{attribute addProperty BoxType "EL9222-4433-0018"}
{attribute addProperty Id "OCP_Inputs_ChannelAT %I*ARRAY[0..1] OF OCP_Inputs_Channel_FE08AF3C6480OCP_Outputs_ChannelAT %Q*ARRAY[0..1] OF OCP_Outputs_Channel_F330A9163240WcStateAT %I*WcState_98A4DF7520.250InfoDataAT %I*InfoData_BC63D37F80100"}
{attribute addProperty CRC "2874621807"}
{attribute addProperty SizeInBites "178"}
{attribute addProperty SizeInBytes "22.25"}
TYPE EL9222_58483589 :
STRUCT
	{attribute addProperty Name "OCP_Inputs_Channel"}
	OCP_Inputs_Channel : ARRAY[0..1] OF OCP_Inputs_Channel_FE08AF3C;
	{attribute addProperty Name "OCP_Outputs_Channel"}
	OCP_Outputs_Channel : ARRAY[0..1] OF OCP_Outputs_Channel_F330A916;
	{attribute addProperty Name "WcState"}
	WcState : WcState_98A4DF75;
	{attribute addProperty Name "InfoData"}
	InfoData : InfoData_BC63D37F;
END_STRUCT
END_TYPE

(* stored: Version 1.2.0.0, ProductVersion 3.1.4024.9
   DUT EL9222_58483589: Id {b635dc54-720d-492f-9bc5-c5c554248e85} *)
